// Mitsubishi GX Works2 project: z04   PLC: Q02/Q02H

PROGRAM MAIN
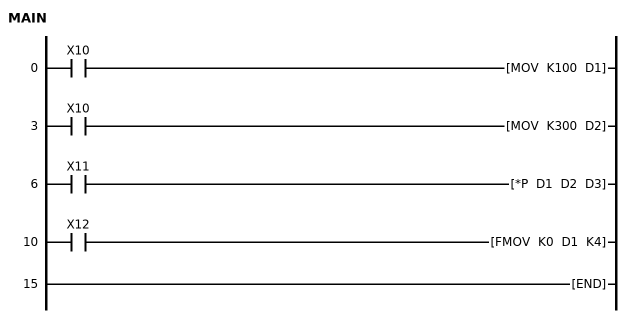
0     LD      X10
      MOV     K100 D1
3     LD      X10
      MOV     K300 D2
6     LD      X11
      *P      D1 D2 D3
10    LD      X12
      FMOV    K0 D1 K4
15    END
END_PROGRAM
